FUNCTION_BLOCK DataTypesString (* Template for an empty basic function block *)
  (* Standard: 61499-2; Description: Normal just propagates the input to the output Internal: sets the output from inside Copyright (c) 2019 Jan Holzweber This program and the accompanying materials are made available under the terms of the Eclipse Public License 2.0 which is available at https://www.eclipse.org/legal/epl-2.0/ SPDX-License-Identifier: EPL-2.0 *)
  (* Version 1.0, 2019-06-05, jholz *)
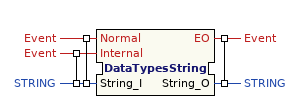
  EVENT_INPUT
    Normal WITH String_I;
    Internal WITH String_I;
  END_EVENT
  EVENT_OUTPUT
    EO WITH String_O;
  END_EVENT
  VAR_INPUT
    String_I : STRING;
  END_VAR
  VAR_OUTPUT
    String_O : STRING;
  END_VAR
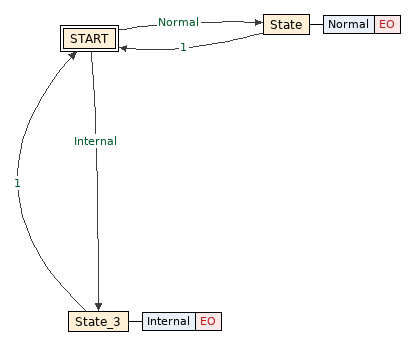
  EC_STATES
    START; (* Initial State *)
    State : Normal -> EO;
    State_3 : Internal -> EO;
  END_STATES
  EC_TRANSITIONS
    START TO State := Normal;
    State TO START := 1;
    START TO State_3 := Internal;
    State_3 TO START := 1;
  END_TRANSITIONS
  ALGORITHM Normal IN ST: (* new algorithm *)
STRING_O:=STRING_I;
  END_ALGORITHM
  ALGORITHM Internal IN ST: (* new algorithm *)
STRING_O:='Setting from Interal';
  END_ALGORITHM
END_FUNCTION_BLOCK
